//     PlcTask Inputs/MAIN.aMovers[6].Axis.Axis.NcToPlc <-> Outputs/ToPlc
//     PlcTask Outputs/MAIN.aMovers[6].Axis.Axis.PlcToNc <-> Inputs/FromPlc
//   Plc/Plc Instance <-> NC-Task 1 SAF/Axes/SimAxis
//     PlcTask Inputs/PRG_Example_Station.fbStationMounting.fbSimAxis.Axis.NcToPlc <-> Outputs/ToPlc
//     PlcTask Outputs/PRG_Example_Station.fbStationMounting.fbSimAxis.Axis.PlcToNc <-> Inputs/FromPlc
//   Plc/Plc Instance <-> NC-Task 1 SAF/Objects/Group1 (CA Group)
//     PlcTask Inputs/MAIN.fbGroup.GroupRef.NcToPlc <-> Group Outputs/ToPLC
//     PlcTask Outputs/MAIN.fbGroup.GroupRef.PlcToNc <-> Group Inputs/FromPLC

CONFIGURATION Plc
    RESOURCE PLC ON TwinCAT3
        TASK PlcTask(INTERVAL := T#10ms, PRIORITY := 20);
        PROGRAM MAIN WITH PlcTask : MAIN;
    END_RESOURCE
END_CONFIGURATION

// ---- POUs/Example Station Implementation/E_StationProcessState.TcDUT
{attribute 'qualified_only'}
{attribute 'strict'}
TYPE E_StationProcessState :
(
	Idle 			:= 0,
	ProcessStart 	:= 1,
	ProcessBusy 	:= 2,
	ProcessDone 	:= 3
);
END_TYPE

// ---- POUs/Example Station Implementation/E_OpMode.TcDUT
{attribute 'qualified_only'}
{attribute 'strict'}
TYPE E_OpMode :
(
	Off := 0,
	Auto := 1,
	Simulation := 2,
	Calibration := 3
);
END_TYPE

// ---- POUs/Example Station Implementation/I_StationProcess.TcIO
INTERFACE I_StationProcess

PROPERTY SetOpMode : E_OpMode
SET
END_SET
END_PROPERTY

PROPERTY State : E_StationProcessState
GET
END_GET
SET
END_SET
END_PROPERTY

METHOD Update
VAR_INPUT
	iStation : I_XTS_Station_PLC;	
END_VAR
END_METHOD

END_INTERFACE

// ---- POUs/MAIN.TcPOU
PROGRAM MAIN
VAR CONSTANT
	N_NBR_MOVERS : USINT := 6;
	N_NBR_STATIONS : USINT := 10;
END_VAR
VAR
	bInitDone, bEnable, bDisable, bStart, bRestart : BOOL;
	bStartSimulation, bStopSimulation : BOOL ;	
	bAllStationsReady : BOOL := TRUE;

	nLoopIndex : UINT;
	iStation : I_XTS_Station;
	bWaitingStation : BOOL;	
	nIndexStationToCommandMoverInto, nIndexStationToMoveAferStart : UINT;


	
	fbSystem		: CHALET_Xts.FB_XTS_System;
	iXtsSystem 		: I_XTS_System_PLC := fbSystem;

	fbEnvironment	: CHALET_Xts.FB_XTS_Environment(ipXtsSystem := fbSystem);
	
	fbGroup			: CHALET_Xts.FB_XTS_Group(ipXtsSystem := fbSystem);
	
	aMovers			: ARRAY[1..N_NBR_MOVERS] OF CHALET_Xts.FB_XTS_Mover(ipXtsSystem := fbSystem);
	
	aStations		: ARRAY[1..N_NBR_STATIONS] OF CHALET_Xts.FB_XTS_Station[
	
												(ipXtsSystem 		:= fbSystem,
												fPositionOnTrack	:= 1750,
												sStationID			:= 'Loading',
												nMoverQueueSize		:= 2,
												fMoverGapAtExit		:= 100,
												fMoverVelocityAtExit:= 500),

												(ipXtsSystem 		:= fbSystem,
												fPositionOnTrack	:= 1950,
												sStationID			:= 'Wait',
												nMoverQueueSize		:= 1,
												fMoverGapAtExit		:= 100,
												fMoverVelocityAtExit:= 500),	

												(ipXtsSystem 		:= fbSystem,
												fPositionOnTrack	:= 2100.54,
												sStationID			:= 'Mounting',
												nMoverQueueSize		:= 1,
												fMoverGapAtExit		:= 200,
												fMoverVelocityAtExit:= 500),
												
												(ipXtsSystem 		:= fbSystem,
												fPositionOnTrack	:= 550,
												sStationID			:= 'Unloading',
												nMoverQueueSize		:= 3,
												fMoverGapAtExit		:= 80,
												fMoverVelocityAtExit:= 500),
												
												(ipXtsSystem 		:= fbSystem,
												fPositionOnTrack	:= 1000,
												sStationID			:= 'WaitBuffer',
												nMoverQueueSize		:= 4,
												fMoverGapAtExit		:= 80,
												fMoverVelocityAtExit:= 200),
	
												(ipXtsSystem 		:= fbSystem,
												fPositionOnTrack	:= 1350,
												sStationID			:= 'WaitLoading',
												nMoverQueueSize		:= 2,
												fMoverGapAtExit		:= 80,
												fMoverVelocityAtExit:= 200),

												(ipXtsSystem		:= fbSystem,
												fPositionOnTrack	:= 1500,
												sStationID			:= 'Trigger1',
												nMoverQueueSize		:= 0,
												fMoverGapAtExit		:= 200,
												fMoverVelocityAtExit:= 500),
												
												(ipXtsSystem		:= fbSystem,
												fPositionOnTrack	:= 2500,
												sStationID			:= 'Trigger2',
												nMoverQueueSize		:= 0,
												fMoverGapAtExit		:= 100,
												fMoverVelocityAtExit:= 200),

												(ipXtsSystem		:= fbSystem,
												fPositionOnTrack	:= 0,
												sStationID			:= 'Trigger3',
												nMoverQueueSize		:= 0,
												fMoverGapAtExit		:= 200,
												fMoverVelocityAtExit:= 500),
												
												(ipXtsSystem 		:= fbSystem,
												fPositionOnTrack	:= 2400,
												sStationID			:= 'Calibration',
												nMoverQueueSize		:= 1,
												fMoverGapAtExit		:= 200,
												fMoverVelocityAtExit:= 500)];										
												
		

	stCommand : CHALET_Xts.Tc3_XTS_Utility.ST_TcIoXtsMoverCommand;
	refCommandHistory : REFERENCE TO ARRAY[1..CHALET_Xts.Tc3_XTS_Utility.TcIoXtsEnvironmentParameterList.MaxMessageCommandHistory] OF CHALET_Xts.Tc3_XTS_Utility.ST_TcIoXtsMoverCommand;

	// change of Gap Control Mode
	bFast, bStandard : BOOL;
	
	// Calibration
	bCalibration : BOOL;												
END_VAR

(*	Todo in a new Tc project:
	- Add Groupe + link
	- StopPositions in XtsStationInfo set to 25 Array
	- Set raillength in groupe
	- Info Server: Stations link
	-
*)

IF NOT bInitDone THEN
	fbSystem.Initialize();
	bInitDone := fbSystem.Initialized;
	iXtsSystem := fbSystem;
	RETURN;
END_IF

// Enabling the System is only possible after a successful Disabling
IF bEnable AND iXtsSystem.Initialized AND iXtsSystem.Disabled THEN
	bEnable := FALSE;	
	iXtsSystem.Enable();
END_IF

// Disabling the System is allways possible
// while E-Stop call disable Methode before cutting 48V
IF bDisable THEN
	bDisable := FALSE;
	iXtsSystem.Disable();
	// set opeationMode to Off
	PRG_Example_Station.setOpMode := E_OpMode.Off;
END_IF

// command all movers into the default station.
IF bStart AND iXtsSystem.Enabled THEN
	// All changes to the dynamic parameters are suppressed, as the start movement is normally slower.
	iXtsSystem.SuppressAllDynamicsChanges := TRUE;	
	bAllStationsReady := FALSE;	

	// delete all Queues
	FOR nLoopIndex := 1 TO N_NBR_STATIONS DO
		aStations[nLoopIndex].DeleteMoversQueue();
	END_FOR

	// send all mover in waiting station and as the next station selct the default station
	nIndexStationToMoveAferStart  := 1;	
	nIndexStationToCommandMoverInto := 5;	
	FOR nLoopIndex := 1 TO N_NBR_MOVERS DO
		aMovers[nLoopIndex].TargedStation := aStations[nIndexStationToCommandMoverInto].LUID;
		aMovers[nLoopIndex].MoveAbsCA(fPosition:=aStations[nIndexStationToCommandMoverInto].PositionOnTrack, fVelocity := 500, fGap := aStations[nIndexStationToCommandMoverInto].StationBehinde.MoverGapAtExit, eDirection := Tc3_Mc3Definitions.MC_DIRECTION.mcDirectionPositive);
		aStations[nIndexStationToCommandMoverInto].AddMoverToQueue(aMovers[nLoopIndex]);
	END_FOR
	
	IF aStations[nIndexStationToCommandMoverInto].AreMoversInPlace THEN
		FOR nLoopIndex := 1 TO N_NBR_MOVERS DO
			aMovers[nLoopIndex].TargedStation := aStations[nIndexStationToMoveAferStart].LUID;
		END_FOR
		
		// set opeationMode to Auto
		PRG_Example_Station.setOpMode := E_OpMode.Auto;
		
		iXtsSystem.SuppressAllDynamicsChanges := FALSE;
		bStart := FALSE;
	END_IF
END_IF	

// 	continue the process after a disable - enable sequence
IF bRestart THEN
	bRestart := FALSE;
	iXtsSystem.SuppressAllDynamicsChanges := FALSE;	
	bAllStationsReady := TRUE;	
	
	FOR nLoopIndex := 1 TO N_NBR_MOVERS DO
		// command the mover with the last command sent 
		aMovers[nLoopIndex].MoveAbsCA(
			fPosition	:= aMovers[nLoopIndex].ParentStation.PositionOnTrack, 
			fVelocity 	:= aMovers[nLoopIndex].LastCmdTargedVelocity,  
			fGap 		:= aMovers[nLoopIndex].LastCmdTargedGap,  
			eDirection 	:= Tc3_Mc3Definitions.MC_DIRECTION.mcDirectionPositive);
	END_FOR
	
	// set opeationMode to Auto
	PRG_Example_Station.setOpMode := E_OpMode.Auto;
END_IF

// set Calibration
IF bCalibration THEN
	bCalibration := FALSE;
	PRG_Example_Station.setOpMode := E_OpMode.Calibration;
END_IF

//Configure AND Start Simulation
IF bStartSimulation THEN
	bStartSimulation := FALSE;
	iXtsSystem.SuppressAllDynamicsChanges := FALSE;	//Enable to adjust Gap + Dynamic depending on Station
	
	iXtsSystem.Station('Loading').	SimulationMode(1.0, 'Mounting');
//	iXtsSystem.Station('Loading').	SimulationMode(0.5, 'Calibration');
//	iXtsSystem.Station('Mounting').	SimulationMode(0.5, 'Unloading');
	iXtsSystem.Station('Unloading').	SimulationMode(1.0, 'Loading');
END_IF

// Stop Simulation
IF bStopSimulation THEN
	bStopSimulation := FALSE;
	FOR nLoopIndex := 1 TO N_NBR_STATIONS DO
		aStations[nLoopIndex].SimulationMode(0,'');
	END_FOR	
	
END_IF

/// replace this section with your Station logic
/// wait for movers, do your process, send the movers to station in front
IF iXtsSystem.Enabled AND bAllStationsReady THEN
	iXtsSystem.SuppressAllDynamicsChanges := FALSE;		
	FOR nLoopIndex := 1 TO N_NBR_STATIONS DO
		//In this aplicationexample, this is an waitingstation
		bWaitingStation := (FIND(aStations[nLoopIndex].LUID,'wait')>0) OR (FIND(aStations[nLoopIndex].LUID,'Wait')>0);		
		//Start process if all movers are in station
		IF aStations[nLoopIndex].AreMoversInPlace AND NOT bWaitingStation THEN
			;
		END_IF
		//Mover is in station and process is done
		IF PRG_Example_Station.fbStationCalib.State = E_StationProcessState.ProcessDone THEN
			//get next station in flow direction who has QueueSize >0 and is not defind as an waiting station(Queuesize >0 but no process)
			iStation := aStations[nLoopIndex].StationsAhead;
			WHILE iStation.MoverQueueSize = 0 OR (FIND(iStation.LUID,'wait')>0) OR (FIND(iStation.LUID,'Wait')>0) DO
				iStation := iStation.StationsAhead;
			END_WHILE

			//send mover in next station
			//XtsSystem.Station(aStations[nLoopIndex].LUID).SendMoversToStation(iStation.LUID);			
		END_IF	
	END_FOR
END_IF


// Changing of Gap Mode for Group (including Control Direction!)
// changes control direction to positiv and mode to fast
IF bFast AND iXtsSystem.Disabled THEN
	bFast := FALSE;
	fbGroup.ChangeGapMode(bFast:= TRUE);
END_IF

	
// changes mode to standard and control direction to both
IF bStandard AND iXtsSystem.Disabled THEN
	bStandard := FALSE;
	fbGroup.ChangeGapMode(bFast:= FALSE);
END_IF

PRG_Example_ProductData();
PRG_Example_Station();

//Update system at the end
fbSystem.Update();

//read command history
refCommandHistory REF= fbSystem.Environment.UtilityEnvirement.XpuTcIo(1).MoverTcIo(1).P_CommandHistory;

//IF XtsSystem.Station('Mounting').AreMoversInPlace THEN
//	XtsSystem.Station('Mounting').MoversInQueue[0].FullAccess.MoveAbsCA(2050,200,500,Tc3_Mc3Definitions.MC_DIRECTION.mcDirectionShortestWay);
//END_IF

END_PROGRAM

// ---- POUs/Example Station Implementation/PRG_Example_Station.TcPOU
PROGRAM PRG_Example_Station
VAR
	bInitDone : BOOL;
	
	fbStationLoad : FB_StationLoadProcess;
	fbStationMounting : FB_StationMoutingProcess;
	fbStationCalib : FB_StationCalibProcess;
	fbStationUnLoad : FB_StationUnLoadProcess;
	
	eOpMode : E_OpMode;
END_VAR

IF NOT bInitDone THEN
	bInitDone := TRUE;
END_IF

//fbStationLoad.Update(iStation := MAIN.iXtsSystem.Station('Loading'));
//fbStationUnLoad.Update(iStation := MAIN.iXtsSystem.Station('Unloading'));
fbStationMounting.Update(iStation := MAIN.iXtsSystem.Station('Mounting'));
fbStationCalib.Update(iStation := MAIN.iXtsSystem.Station('Calibration'));

fbStationLoad.SetOpMode 	:= PRG_Example_Station.eOpMode;
fbStationMounting.SetOpMode := PRG_Example_Station.eOpMode;
fbStationCalib.SetOpMode 	:= PRG_Example_Station.eOpMode;
fbStationUnLoad.SetOpMode	:= PRG_Example_Station.eOpMode;

METHOD CmdOpMode
VAR_INPUT
END_VAR
END_METHOD

PROPERTY setOpMode : E_OpMode
SET
PRG_Example_Station.eOpMode := setOpMode;
END_SET
END_PROPERTY

END_PROGRAM

// ---- POUs/Example Station Implementation/FB_StationLoadProcess.TcPOU
FUNCTION_BLOCK FB_StationLoadProcess EXTENDS FB_StationBase
VAR
END_VAR

METHOD Update
VAR_INPUT
	iStation : I_XTS_Station_PLC;
END_VAR
VAR_INST
	fbTonDelay : ton;
END_VAR
SUPER^.Update(iStation := iStation);

CASE nState OF
	E_StationProcessState.Idle:
		;
		
	E_StationProcessState.ProcessStart:
		CASE eOpMode OF
			E_OpMode.Auto:
				nState := E_StationProcessState.ProcessBusy;
			E_OpMode.Calibration:
				nState := E_StationProcessState.ProcessDone;	// go ahead to Station Calibration
		END_CASE
		
	E_StationProcessState.ProcessBusy:
		fbTonDelay(In:= TRUE, PT:= T#250MS);
		IF fbTonDelay.Q THEN
			fbTonDelay(In:= FALSE);
			nState := E_StationProcessState.ProcessDone;			
		END_IF
		
	E_StationProcessState.ProcessDone:
		CASE eOpMode OF
			E_OpMode.Simulation:
				; // wait nothing to do
			E_OpMode.Auto:
				main.iXtsSystem.Station('Loading').SendMoversToStation('Mounting');
			E_OpMode.Calibration:
				main.iXtsSystem.Station('Loading').SendMoversToStation('Calibration');
		END_CASE;
END_CASE
END_METHOD

END_FUNCTION_BLOCK

// ---- POUs/Example Station Implementation/FB_StationBase.TcPOU
FUNCTION_BLOCK FB_StationBase IMPLEMENTS I_StationProcess
VAR
	nState : E_StationProcessState;
	nStep : INT;
	eOpMode : E_OpMode;	
END_VAR

PROPERTY SetOpMode : E_OpMode
SET
eOpMode := SetOpMode;
END_SET
END_PROPERTY

PROPERTY State : E_StationProcessState
GET
State := nState;
END_GET
SET
nState := State;
END_SET
END_PROPERTY

METHOD Update
VAR_INPUT
	iStation : I_XTS_Station_PLC;
END_VAR
VAR_INST
	fbTriggerMoverInPlace : R_TRIG; 
END_VAR
//This is executed once when the mover arrives at the station
fbTriggerMoverInPlace(CLK:= iStation.AreMoversInPlace);
IF fbTriggerMoverInPlace.Q THEN
	State := E_StationProcessState.ProcessStart;
END_IF
IF iStation.AreMoversInPlace = FALSE THEN
	State := E_StationProcessState.Idle;
END_IF
END_METHOD

END_FUNCTION_BLOCK

// ---- POUs/Example Station Implementation/FB_StationMoutingProcess.TcPOU
FUNCTION_BLOCK FB_StationMoutingProcess EXTENDS FB_StationBase
VAR
	bInitDone : BOOL;
	fbSimAxis : CHALET_Nc.FB_NcAxis;
	iTempAxis : I_NcAxis_PLC;
	nAxisId : UDINT;

	iFeedback : I_CH_Feedback;
	hr : HRESULT;
	
	fbTonP1 : TON;
	fbTonP2 : TON;
	fbTonP3 : TON;

END_VAR

METHOD Update
VAR_INPUT
	iStation : I_XTS_Station_PLC;
END_VAR
VAR
	iTempMover : I_XTS_Mover;
END_VAR
VAR_INST
	fbTriggerMoverInPlace : R_TRIG; 
END_VAR
//This is executed once when the mover arrives at the station
fbTriggerMoverInPlace(CLK:= iStation.AreMoversInPlace);
IF fbTriggerMoverInPlace.Q THEN
	State := E_StationProcessState.ProcessStart;
END_IF

IF bInitDone = FALSE THEN
	fbSimAxis.Initialize();
	bInitDone := 	fbSimAxis.Initialized;					
	RETURN;
END_IF

IF fbSimAxis.MotionState = MC_AxisStates.MC_AXISSTATE_DISABLED THEN
	fbSimAxis.PowerOn();
END_IF

fbSimAxis.Update();


CASE nState OF
	E_StationProcessState.Idle:
		;
		
	E_StationProcessState.ProcessStart:
		fbSimAxis.SetActPosition(0);
		nAxisId := MAIN.iXtsSystem.Station('Mounting').MoversInQueue[0].FullAccess.getAxisRef.NcToPlc.AxisId;
		nState := E_StationProcessState.ProcessBusy;
		
	E_StationProcessState.ProcessBusy:
		CASE nStep OF 
			
			0: // gearIn
				iFeedback := Main.aMovers[nAxisId].Axis.GearIn(
					ipMasterAxisAdapter := fbSimAxis, 
					fRatioNumerator := 1, 
					nRatioDenominator := 1, 
					fAcceleration := MC_DEFAULT, 
					fDeceleration := MC_DEFAULT, 
					fJerk := MC_DEFAULT);
				
					IF iFeedback.Done OR iFeedback.Busy THEN
						nStep:= nStep + 1;					
					END_IF
				
			1: // wait for done
				IF iFeedback.Done THEN
					nStep:= nStep + 1;										
				END_IF
			
			2 : // wait for P1
				fbTonP1.IN := TRUE;
				IF fbTonP1.Q THEN
					fbTonP1.IN := FALSE;
					nStep:= nStep + 1;
				END_IF
				
			3 : // move forward to P2
				iFeedback := fbSimAxis.MoveAbsolute(
					fPosition := 50, 
					fVelocity := 500, 
					fAcceleration := 2000, 
					fDeceleration := 2000, 
					fJerk := 5000, 
					eBufferMode := MC_Aborting);
					
				IF iFeedback.Busy OR iFeedback.Done THEN
					nStep:= nStep + 1;					
				END_IF
				
			4: // wait for done
				IF iFeedback.Done THEN
					nStep:= nStep + 1;										
				END_IF
				
			5: // wait for P2
				fbTonP2.IN := TRUE;
				IF fbTonP2.Q THEN
					fbTonP2.IN := FALSE;
					nStep:= nStep + 1;
				END_IF
				
			6 : // move backward to P3
				iFeedback := fbSimAxis.MoveAbsolute(
					fPosition := -50, 
					fVelocity := 500, 
					fAcceleration := 2000, 
					fDeceleration := 2000, 
					fJerk := 5000, 
					eBufferMode := MC_Aborting);
					
				IF iFeedback.Busy OR iFeedback.Done THEN
					nStep:= nStep + 1;					
				END_IF
				
			7: // wait for done
				IF iFeedback.Done THEN
					nStep:= nStep + 1;										
				END_IF
				
			8: // wait for P3
				fbTonP3.IN := TRUE;
				IF fbTonP3.Q THEN
					fbTonP3.IN := FALSE;
					nStep:= nStep + 1;
				END_IF
				
			9: // gearOut
				iFeedback := Main.aMovers[nAxisId].Axis.GearOut();
					
				IF iFeedback.Busy OR iFeedback.Done THEN
					nStep:= nStep + 1;
				END_IF
			
			10: // wait for done
				hr := Main.aMovers[nAxisId].Axis.Feedback.HR;
				IF checkOK(hr) THEN
					nStep:= nStep + 1;										
				END_IF
				
			11: // done
				nStep:= 0;
				nState := E_StationProcessState.ProcessDone;
				
		END_CASE
				
	E_StationProcessState.ProcessDone:
		IF __QUERYINTERFACE(MAIN.aMovers[nAxisId], iTempMover) THEN
			iTempMover.TargedStation := 'Unloading';
		END_IF
		nState := E_StationProcessState.Idle;
END_CASE

fbTonP1(PT:= T#100MS);
fbTonP2(PT:= T#250MS);
fbTonP3(PT:= T#300MS);
END_METHOD

END_FUNCTION_BLOCK

// ---- POUs/Example Station Implementation/FB_StationCalibProcess.TcPOU
FUNCTION_BLOCK FB_StationCalibProcess EXTENDS FB_StationBase
VAR
	fbTonSettling : TON;
	fbRandomValue : DRAND;
	aPosCorrLim : ARRAY[1..MAIN.N_NBR_MOVERS] OF TC2_MC2.MC_PositionCorrectionLimiter;
	
	nDist AT%I*: UINT;
//	aBuffer : ARRAY[1..1000] OF UINT;
	nCnt : INT;
//	iAvg : UDINT;
	nAfterCalibration : UINT;
	
	bInitDone : BOOL;
	fbMovingAvg : FB_CTRL_MOVING_AVERAGE;
	stParams : ST_CTRL_MOVING_AVERAGE_PARAMS;
	aData : ARRAY[0..100] OF LREAL;
END_VAR

METHOD Initialize : BOOL
VAR_INPUT
END_VAR
stParams.nSamplesToFilter := 100;
stParams.nWorkArray_SIZEOF := SIZEOF(aData);
stParams.pWorkArray_ADR := ADR(aData);
stParams.tCtrlCycleTime := UDINT_TO_TIME(_TaskInfo[GETCURTASKINDEXEX()].CycleTime)/10000;
stParams.tTaskCycleTime := UDINT_TO_TIME(_TaskInfo[GETCURTASKINDEXEX()].CycleTime)/10000;

fbMovingAvg.eMode := E_CTRL_MODE.eCTRL_MODE_ACTIVE;
fbMovingAvg(stParams := stParams);

Initialize := TRUE;
END_METHOD

METHOD Update
VAR_INPUT
	iStation : I_XTS_Station_PLC;
END_VAR
VAR
	iMoverTemp : I_XTS_Mover;
END_VAR
IF bInitDone = FALSE THEN
	bInitDone := Initialize();
END_IF

SUPER^.Update(iStation := iStation);

CASE nState OF
	E_StationProcessState.Idle:
		;
		
	E_StationProcessState.ProcessStart:
		fbTonSettling.IN := TRUE;
		IF fbTonSettling.Q THEN
			fbTonSettling.IN := FALSE;
			nState := E_StationProcessState.ProcessBusy;
		END_IF

		
	E_StationProcessState.ProcessBusy:
		// get Mover
		IF __QUERYINTERFACE(MAIN.iXtsSystem.Station('Calibration').MoversInQueue[0], iMoverTemp) THEN
			aPosCorrLim[iMoverTemp.getAxisRef.DriveAddress.NcAxisId](
				Axis:= iMoverTemp.getAxisRef,  
				CorrectionMode:= E_AxisPositionCorrectionMode.POSITIONCORRECTION_MODE_FAST, 
				Acceleration:= 1000);	
		END_IF


		CASE nStep OF 
			0: // reset to 0 if active correction
				IF aPosCorrLim[iMoverTemp.getAxisRef.DriveAddress.NcAxisId].Busy THEN
					aPosCorrLim[iMoverTemp.getAxisRef.DriveAddress.NcAxisId].PositionCorrectionValue := 0;
					aPosCorrLim[iMoverTemp.getAxisRef.DriveAddress.NcAxisId].Enable := TRUE;
					IF aPosCorrLim[iMoverTemp.getAxisRef.DriveAddress.NcAxisId].Busy AND aPosCorrLim[iMoverTemp.getAxisRef.DriveAddress.NcAxisId].Limiting OR aPosCorrLim[iMoverTemp.getAxisRef.DriveAddress.NcAxisId].PositionCorrectionValue <= 0.1 THEN
						nStep:= nStep + 1;
					END_IF
				ELSE
					nStep:= nStep + 1;
				END_IF

			1: // wait for correction is set to 0
				IF aPosCorrLim[iMoverTemp.getAxisRef.DriveAddress.NcAxisId].Limiting =FALSE THEN
					nCnt := 1;
					nStep:= nStep + 1;
				END_IF

			2: // wait for setteling
				fbTonSettling.IN := TRUE;
				fbMovingAvg.eMode := e_Ctrl_Mode.eCTRL_MODE_RESET;
				IF fbTonSettling.Q THEN
					fbTonSettling.IN := FALSE;
					nStep:= nStep + 1;
				END_IF
				
			3: // Set Mode to Active
				fbMovingAvg.eMode := e_Ctrl_Mode.eCTRL_MODE_ACTIVE;
				IF fbMovingAvg.eState = E_CTRL_STATE.eCTRL_STATE_ACTIVE THEN
					nStep:= nStep + 1;
				END_IF
			
			4:
				{IF defined (HW_Lyssach)}
					IF nDist >= 1000 AND nDist <=2000 THEN // validate measurement value
						fbMovingAvg.fIn := nDist;
					ELSE
						fbMovingAvg.fIn := 1280;
					END_IF
					fbMovingAvg(stParams := stParams);
					nCnt := nCnt + 1;
					IF nCnt > 100 THEN
						nStep:= nStep + 1;
					END_IF
				{ELSE}		
					fbRandomValue(Seed:= UDINT_TO_INT(_TaskInfo[GETCURTASKINDEXEX()].CycleCount));
					nStep:= nStep + 1;
				{END_IF}
				
				
			5: // set correction
				{IF defined (HW_Lyssach)}
					aPosCorrLim[iMoverTemp.getAxisRef.DriveAddress.NcAxisId].PositionCorrectionValue := 128.0-fbMovingAvg.fOut/10.0;
				{ELSE}
					aPosCorrLim[iMoverTemp.getAxisRef.DriveAddress.NcAxisId].PositionCorrectionValue := (fbRandomValue.Num-0.5)*20;
				{END_IF}
				aPosCorrLim[iMoverTemp.getAxisRef.DriveAddress.NcAxisId].Enable := TRUE;
				IF aPosCorrLim[iMoverTemp.getAxisRef.DriveAddress.NcAxisId].Busy AND aPosCorrLim[iMoverTemp.getAxisRef.DriveAddress.NcAxisId].Limiting OR aPosCorrLim[iMoverTemp.getAxisRef.DriveAddress.NcAxisId].PositionCorrectionValue <= 0.1 THEN
					nStep:= nStep + 1;
				END_IF
				
			6: // wait for correction done
				fbMovingAvg.eMode := E_CTRL_MODE.eCTRL_MODE_IDLE;
				IF aPosCorrLim[iMoverTemp.getAxisRef.DriveAddress.NcAxisId].Limiting =FALSE THEN
					nStep:= nStep + 1;
				END_IF
				
			7: // wait for setteling
				fbTonSettling.IN := TRUE;
				IF fbTonSettling.Q THEN
					nAfterCalibration := nDist;
					fbTonSettling.IN := FALSE;
					nStep:= 0;
					nState := E_StationProcessState.ProcessDone;
				END_IF
		END_CASE
		
	E_StationProcessState.ProcessDone:
		main.iXtsSystem.Station('Calibration').SendMoversToStation('WaitBuffer');

END_CASE

fbTonSettling(PT:= T#500MS);
END_METHOD

END_FUNCTION_BLOCK

// ---- POUs/Example Station Implementation/FB_StationUnLoadProcess.TcPOU
FUNCTION_BLOCK FB_StationUnLoadProcess EXTENDS FB_StationBase
VAR
END_VAR

METHOD Update
VAR_INPUT
	iStation : I_XTS_Station_PLC;
END_VAR
VAR_INST
	fbTonDelay : ton;
END_VAR
SUPER^.Update(iStation := iStation);

CASE nState OF
	E_StationProcessState.Idle:
		;
		
	E_StationProcessState.ProcessStart:
		nState := E_StationProcessState.ProcessBusy;
		
	E_StationProcessState.ProcessBusy:
		fbTonDelay(In:= TRUE, PT:= T#250MS);
		IF fbTonDelay.Q THEN
			fbTonDelay(In:= FALSE);
			nState := E_StationProcessState.ProcessDone;			
		END_IF
		
	E_StationProcessState.ProcessDone:
		CASE eOpMode OF
			E_OpMode.Simulation:
				; // wait nothing to do
			E_OpMode.Auto, E_OpMode.Calibration:
				main.iXtsSystem.Station('Unloading').SendMoversToStation('Loading');
		END_CASE;
END_CASE
END_METHOD

END_FUNCTION_BLOCK

// ---- POUs/Example Product Data/PRG_Example_ProductData.TcPOU
PROGRAM PRG_Example_ProductData
VAR
	bInitDone : BOOL;
		
	aProductsFormatA 	: ARRAY[0..(MAIN.N_NBR_MOVERS-1)] OF FB_ProductDataA;
	fbProductsUnused 	: CHALET_BaseComponents.FB_CH_List; //In this example this list is used to transfer products to the XTS
	fbProductsOnMover 	: CHALET_BaseComponents.FB_CH_List; //As long as the products are on the XTS, each of them can be reached via this list and the interface to the mover can also be requested.
	
	ipObject 			: I_CH_Object;
	ipProductFormatA 	: I_ProductDataA;

	ipStationLoad, ipStationModify, ipStationUnload : I_XTS_Station_PLC;
	fbTriggerMoverInPlace1, fbTriggerMoverInPlace2, fbTriggerMoverInPlace3 : R_TRIG; 
	
	nIdx : UDINT;
END_VAR

IF NOT bInitDone THEN
	bInitDone := TRUE;
	
	//Put all product informations in a list to easy access them
	FOR nIdx := 0 TO (MAIN.N_NBR_MOVERS-1) DO
		fbProductsUnused.AddObject(aProductsFormatA[nIdx]);
	END_FOR
END_IF



//Station A: put empty product info FB on mover
ipStationLoad := MAIN.iXtsSystem.Station('Loading');
//This is executed once when the mover arrives at the station
fbTriggerMoverInPlace1(CLK:= ipStationLoad.AreMoversInPlace);
IF fbTriggerMoverInPlace1.Q THEN
	//Do this for each mover inside the station
	FOR nIdx := 0 TO (ipStationLoad.MoverQueueSize-1) DO
		
		// Only execute if datacontainer on mover is empty
		IF ipStationLoad.MoversInQueue[nIdx].ProductData = 0 THEN
			
			//Get an unused product OR handover here the product data from the previous process step here
			ipObject := fbProductsUnused.GetRandomObject();
			
			//Remove an put in OnMovers List
			fbProductsUnused.RemoveObject(ipObject);
			fbProductsOnMover.AddObject(ipObject);
			
			
			//Query whether the FB behind this instance implements the following interface and get it.
			IF __QUERYINTERFACE(ipObject, ipProductFormatA) THEN		
				//Store the interface in the Mover
				ipStationLoad.MoversInQueue[nIdx].ProductData := ipProductFormatA; // <= one of the important steps. Everything else around is application specific
			END_IF
		
		END_IF
		

	END_FOR
END_IF


//Station B: read/write product info 
ipStationModify := MAIN.iXtsSystem.Station('Mounting');
//This is executed once when the mover arrives at the station
fbTriggerMoverInPlace2(CLK:= ipStationModify.AreMoversInPlace);
IF fbTriggerMoverInPlace2.Q THEN
	//Do this for each mover inside the station
	FOR nIdx := 0 TO (ipStationModify.MoverQueueSize-1) DO
		
		//Query whether the FB behind this instance implements the following interface and get it.
		IF __QUERYINTERFACE(ipStationModify.MoversInQueue[nIdx].ProductData, ipProductFormatA) THEN // <= one of the important steps. Everything else around is application specific
			ipProductFormatA.Data.nQuality := (ipProductFormatA.Data.nQuality + 42)MOD 100;	
			ipProductFormatA.Data.bGoodProduct := ipProductFormatA.Data.nQuality >= 80;
		END_IF
	
	END_FOR
END_IF



//Station C: Remove Produkt from XTS
ipStationUnload := MAIN.iXtsSystem.Station('Unloading');
//This is executed once when the mover arrives at the station
fbTriggerMoverInPlace3(CLK:= ipStationUnload.AreMoversInPlace);
IF fbTriggerMoverInPlace3.Q THEN
	//Do this for each mover inside the station
	FOR nIdx := 0 TO (ipStationUnload.MoverQueueSize-1) DO
		
		//Query whether the FB behind this instance implements the following interface and get it.
		IF __QUERYINTERFACE(ipStationUnload.MoversInQueue[nIdx].ProductData, ipObject) THEN
			
			//Handover to next processing unit OR in this case, put in UnusedList
			fbProductsOnMover.RemoveObject(ipObject);
			fbProductsUnused.AddObject(ipObject);
		END_IF
		
		// Clear mover storage
		ipStationUnload.MoversInQueue[nIdx].ProductData := 0; // <= one of the important steps. Everything else around is application specific
	END_FOR
END_IF

END_PROGRAM

// ---- POUs/Example Product Data/FB_ProductDataA.TcPOU
FUNCTION_BLOCK FB_ProductDataA EXTENDS FB_XTS_ProductData IMPLEMENTS I_ProductDataA
VAR
	stData 	: ST_ProductDataA;
END_VAR

{attribute 'monitoring':='call'}
PROPERTY Data : REFERENCE TO ST_ProductDataA
GET
Data REF= stData;
END_GET
END_PROPERTY

END_FUNCTION_BLOCK

// ---- VISUs/Visualization.TcVIS
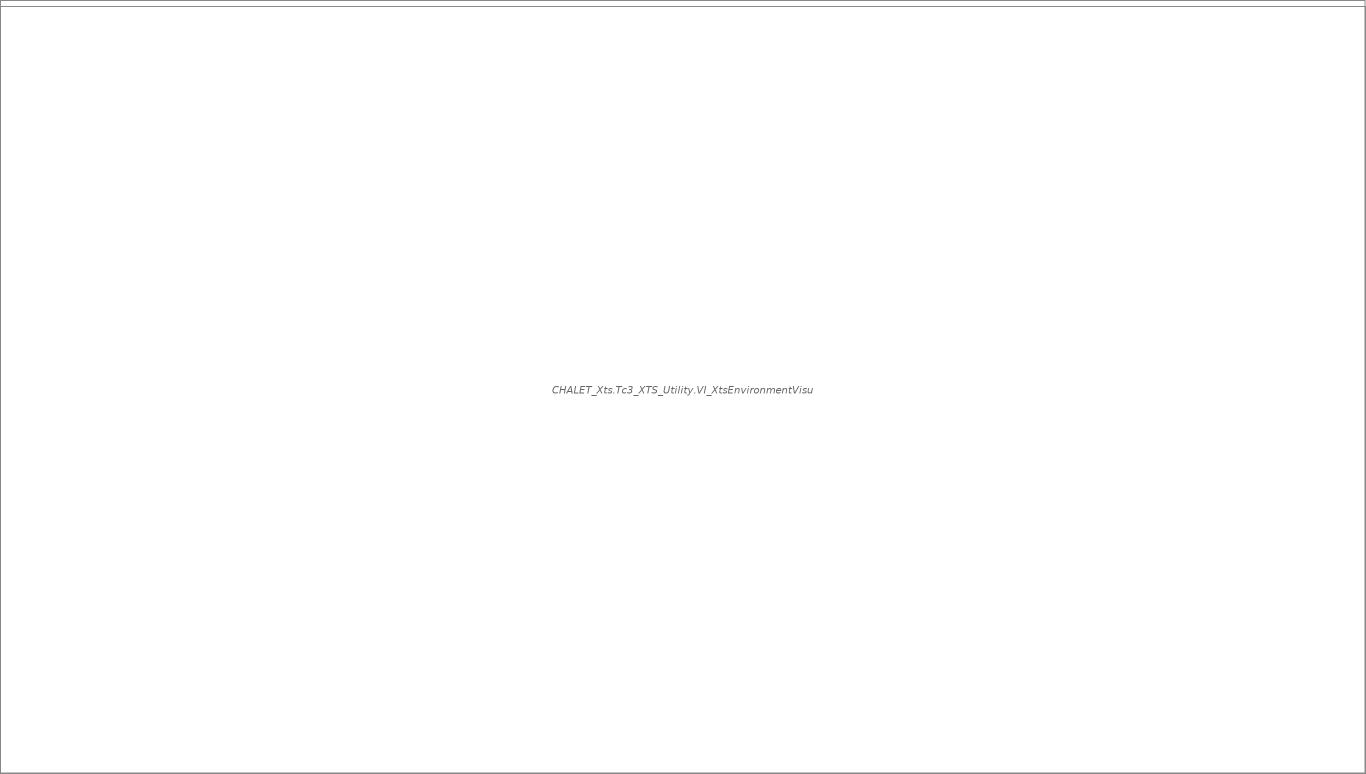
VISUALIZATION Visualization  // 1366x774
    Frame (0,6 1366x768)
        shows CHALET_Xts.Tc3_XTS_Utility.VI_XtsEnvironmentVisu()
END_VISUALIZATION
